TYPE UNI_HMI_WheelHouseInput2 :
UNION
	arWheelHouseInput : ARRAY[1..400] OF BOOL;
	List :ST_WheelhouseInput;
END_UNION
END_TYPE

(* stored: Version 1.1.0.1, ProductVersion 3.1.4024.13
   DUT UNI_HMI_WheelHouseInput2: Id {8a399633-ee5d-47d8-bf0b-a247d912cf19} *)
